RoboDK station: myUR3.rdk

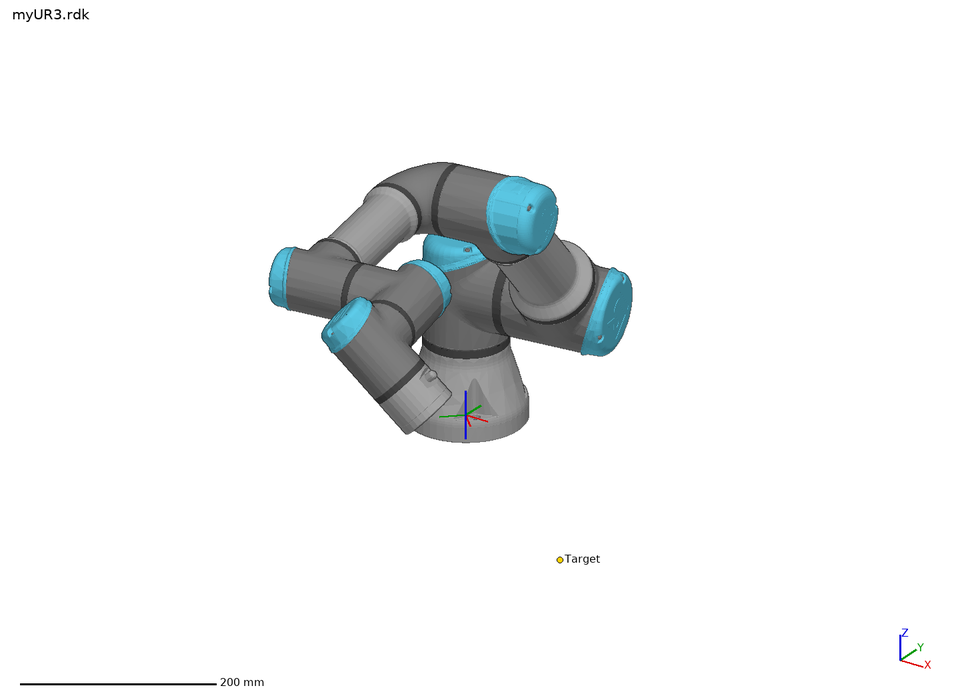
[picture v0: the station drawn from its stored meshes, robots at their saved joint values, targets as dots, program paths as lines]
Station myUR3 (saved by RoboDK 5.6.8). Poses are relative to the parent item; angles as X-Y-Z fixed-axis rotations.
  - frame UR3e Base at (0, 0, 0) mm
    - robot UR3e: 6 axes, payload 3 kg, reach 500 mm, repeatability 0.03 mm, weight 11 kg
        modified DH rows (alpha deg, a mm, theta deg, d mm): 0, 0, 0, 151.9; 90, 0, 180, 0; 0, 243.55, 0, 0; 0, 213.2, 0, 131.05; -90, 0, 0, 85.35; 90, 0, 180, 92.1
        joint limits [-360, -360, -360, -360, -360, -360] to [360, 360, 360, 360, 360, 360]; home [0, -90, -90, 0, 90, 0]; saved at [97.375, -47.164, 50.585, -85.863, -45.504, -100.721]
      - tool Tool 1, TCP at (0, 0, 200) mm
    - frame B0 frame at (0, 0, 0) mm, rotated rx 180 ry 0 rz -45 deg
      - target Target (Cartesian target) at (550, 0, -100) mm, rotated rx 45 ry 0 rz 30 deg; joints [135, -90, 90, -90, -90, -90] of UR3e
  - program My Prog (1 instructions, listed below)

--- program My Prog (robot UR3e) ---
  MoveJ (Target)
